FUNCTION_BLOCK PUBLIC PAEScaleGravimetric EXTENDS PAEScaleBase IMPLEMENTS IPAScaleGravimetric
VAR_INPUT
END_VAR
VAR_OUTPUT
END_VAR
VAR
	_CalmingTime : TIME;
	_CalmingWeight : LREAL;
	_IsDischarging : BOOL;
	_IsManualDosing : BOOL;
	_IsTared : BOOL;
	_ReqZeroReset : BOOL;
	_ReqZeroSet : BOOL;
	_StoredTareWeight : LREAL;
	_TareWeight : LREAL;
	_ZeroSet : BOOL;
	_ReqIsTared : BOOL;
	_TareCounterReq : DINT;
	_ActualWeightExternal : LREAL;
	_TareCounterRes : DINT;
END_VAR

{attribute 'monitoring' := 'call'}
//{attribute 'TcRpcEnable'}
PROPERTY PUBLIC ActualWeightExternal : LREAL
GET
ActualWeightExternal := _ActualWeightExternal;
END_GET
SET
_ActualWeightExternal := ActualWeightExternal;
Root.OnPropertyChangedLReal(THIS^, 84, _ActualWeightExternal);
END_SET
END_PROPERTY

{attribute 'monitoring' := 'call'}
//{attribute 'TcRpcEnable'}
PROPERTY PUBLIC CalmingTime : TIME
GET // PUBLIC
CalmingTime := _CalmingTime;
END_GET
SET // PUBLIC
_CalmingTime := CalmingTime;
Root.OnPropertyChangedTime(THIS^, 72, _CalmingTime);
END_SET
END_PROPERTY

{attribute 'monitoring' := 'call'}
//{attribute 'TcRpcEnable'}
PROPERTY CalmingWeight : LREAL
GET
CalmingWeight := _CalmingWeight;
END_GET
SET
_CalmingWeight := CalmingWeight;
Root.OnPropertyChangedLReal(THIS^, 73, _CalmingWeight);
END_SET
END_PROPERTY

METHOD FB_postinit
VAR_INPUT
	root : IACVariobatch;
END_VAR
SUPER^.FB_postinit(root);
root.OnPropertyChangedTime(THIS^, 72, _CalmingTime);
root.OnPropertyChangedLReal(THIS^, 73, _CalmingWeight);
root.OnPropertyChangedBool(THIS^,74, _ReqZeroSet);
root.OnPropertyChangedBool(THIS^, 75, _ReqZeroReset);
root.OnPropertyChangedLReal(THIS^, 76, _TareWeight);
root.OnPropertyChangedLReal(THIS^, 77, _StoredTareWeight);
root.OnPropertyChangedBool(THIS^, 78, _IsDischarging);
root.OnPropertyChangedBool(THIS^, 79, _IsTared);
root.OnPropertyChangedBool(THIS^, 80, _ZeroSet);
root.OnPropertyChangedBool(THIS^, 81, _IsManualDosing);
root.OnPropertyChangedBool(THIS^, 82, _ReqIsTared);
root.OnPropertyChangedDInt(THIS^, 83, _TareCounterReq);
root.OnPropertyChangedLReal(THIS^, 84, _ActualWeightExternal);
root.OnPropertyChangedDInt(THIS^, 85, _TareCounterRes);
END_METHOD

METHOD PUBLIC InvokeSetterBool
VAR_INPUT
	PropertyID : INT;
	PropertyValue : BOOL;
END_VAR
SUPER^.InvokeSetterBool(PropertyID, PropertyValue);
CASE PropertyID OF
	74:
		ReqZeroSet := PropertyValue;
	75:
		ReqZeroReset := PropertyValue;
	78:
		IsDischarging := PropertyValue;
	79:
		IsTared := PropertyValue;
	80:
		ZeroSet := PropertyValue;
	81:
		IsManualDosing := PropertyValue;
	82:
		ReqIsTared := PropertyValue;
END_CASE
END_METHOD

METHOD PUBLIC InvokeSetterDInt
VAR_INPUT
	PropertyID : INT;
	PropertyValue : DINT;
END_VAR
SUPER^.InvokeSetterDInt(PropertyID, PropertyValue);
CASE PropertyID OF
	83:
		TareCounterReq := PropertyValue;
	85:
		TareCounterRes := PropertyValue;
END_CASE
END_METHOD

METHOD PUBLIC InvokeSetterLReal
VAR_INPUT
	PropertyID : INT;
	PropertyValue : LREAL;
END_VAR
SUPER^.InvokeSetterLReal(PropertyID, PropertyValue);
CASE PropertyID OF
	73:
		CalmingWeight := PropertyValue;
	76:
		TareWeight := PropertyValue;
	77:
		StoredTareWeight := PropertyValue;
	84:
		ActualWeightExternal := PropertyValue;
END_CASE
END_METHOD

METHOD PUBLIC InvokeSetterTime
VAR_INPUT
	PropertyID : INT;
	PropertyValue : DINT;
END_VAR
SUPER^.InvokeSetterTime(PropertyID, PropertyValue);
CASE PropertyID OF 
	72:
		CalmingTime := TO_TIME(PropertyValue);
END_CASE
END_METHOD

{attribute 'monitoring' := 'call'}
//{attribute 'TcRpcEnable'}
PROPERTY PUBLIC IsDischarging : BOOL
GET // PUBLIC
IsDischarging := _IsDischarging;
END_GET
SET // PUBLIC
_IsDischarging := IsDischarging;
Root.OnPropertyChangedBool(THIS^, 78, _IsDischarging);
END_SET
END_PROPERTY

METHOD PUBLIC IsEnabledResetZero : BOOL
VAR_INPUT
END_VAR
END_METHOD

METHOD PUBLIC IsEnabledSetZero : BOOL
VAR_INPUT
END_VAR
END_METHOD

{attribute 'monitoring' := 'call'}
//{attribute 'TcRpcEnable'}
PROPERTY PUBLIC IsManualDosing : BOOL
GET // PUBLIC
IsManualDosing := _IsManualDosing;
END_GET
SET // PUBLIC
_IsManualDosing := IsManualDosing;
Root.OnPropertyChangedBool(THIS^, 81, _IsManualDosing);
END_SET
END_PROPERTY

{attribute 'monitoring' := 'call'}
//{attribute 'TcRpcEnable'}
PROPERTY PUBLIC IsTared : BOOL
GET // PUBLIC
IsTared := _IsTared;
END_GET
SET // PUBLIC
_IsTared := IsTared;
Root.OnPropertyChangedBool(THIS^, 79, _IsTared);
END_SET
END_PROPERTY

METHOD OnInitMemory
VAR_INPUT
	root : IACVariobatch;
END_VAR
RegisterProperty(root, 72, GCL.cSizeTIME); //CalmingTime
RegisterProperty(root, 73, GCL.cSizeLREAL); //CalmingWeight
RegisterProperty(root, 74, GCL.cSizeBYTE); //ReqZeroSet
RegisterProperty(root, 75, GCL.cSizeBYTE); //ReqZeroReset
RegisterProperty(root, 76, GCL.cSizeLREAL); //TareWeight
RegisterProperty(root, 77, GCL.cSizeLREAL); //StoredTaredWeight
RegisterProperty(root, 78, GCL.cSizeBYTE); //IsDischarging
RegisterProperty(root, 79, GCL.cSizeBYTE); //IsTared
RegisterProperty(root, 80, GCL.cSizeBYTE); //ZeroSet
RegisterProperty(root, 81, GCL.cSizeBYTE); //IsManualDosing
RegisterProperty(root, 82, GCL.cSizeBYTE); //ReqIsTared
RegisterProperty(root, 83, GCL.cSizeDINT); //TareCounterReq
RegisterProperty(root, 84, GCL.cSizeLREAL); //ActualWeightExternal
RegisterProperty(root, 85, GCL.cSizeDINT); //TareCounterRes
SUPER^.OnInitMemory(root);
END_METHOD

{attribute 'monitoring' := 'call'}
//{attribute 'TcRpcEnable'}
PROPERTY PUBLIC ReqIsTared : BOOL
GET
ReqIsTared := _ReqIsTared;
END_GET
SET // PUBLIC
_ReqIsTared := ReqIsTared;
Root.OnPropertyChangedBool(THIS^, 82, _ReqIsTared);
END_SET
END_PROPERTY

{attribute 'monitoring' := 'call'}
//{attribute 'TcRpcEnable'}
PROPERTY PUBLIC ReqZeroReset : BOOL
GET // PUBLIC
ReqZeroReset := _ReqZeroReset;
END_GET
SET // PUBLIC
_ReqZeroReset := ReqZeroReset;	
Root.OnPropertyChangedBool(THIS^, 75, _ReqZeroReset);
END_SET
END_PROPERTY

{attribute 'monitoring' := 'call'}
//{attribute 'TcRpcEnable'}
PROPERTY PUBLIC ReqZeroSet : BOOL
GET // PUBLIC
ReqZeroSet := _ReqZeroSet;
END_GET
SET // PUBLIC
_ReqZeroSet := ReqZeroSet;	
Root.OnPropertyChangedBool(THIS^,74, _ReqZeroSet);
END_SET
END_PROPERTY

METHOD PUBLIC ResetZero
VAR_INPUT
END_VAR
END_METHOD

METHOD PUBLIC SetZero
VAR_INPUT
END_VAR
END_METHOD

{attribute 'monitoring' := 'call'}
//{attribute 'TcRpcEnable'}
PROPERTY PUBLIC StoredTareWeight : LREAL
GET // PUBLIC
StoredTareWeight := _StoredTareWeight;
END_GET
SET // PUBLIC
_StoredTareWeight := StoredTareWeight;
Root.OnPropertyChangedLReal(THIS^, 77, _StoredTareWeight);
END_SET
END_PROPERTY

{attribute 'monitoring' := 'call'}
//{attribute 'TcRpcEnable'}
PROPERTY PUBLIC TareCounterReq : DINT
GET
TareCounterReq := _TareCounterReq;
END_GET
SET
_TareCounterReq := TareCounterReq;
Root.OnPropertyChangedDInt(THIS^, 83, _TareCounterReq);
END_SET
END_PROPERTY

{attribute 'monitoring' := 'call'}
//{attribute 'TcRpcEnable'}
PROPERTY PUBLIC TareCounterRes : DINT
GET
TareCounterRes := _TareCounterRes;
END_GET
SET
_TareCounterRes := TareCounterRes;
Root.OnPropertyChangedDInt(THIS^, 85, _TareCounterRes);
END_SET
END_PROPERTY

{attribute 'monitoring' := 'call'}
//{attribute 'TcRpcEnable'}
PROPERTY PUBLIC TareWeight : LREAL
GET // PUBLIC
TareWeight := _TareWeight;
END_GET
SET // PUBLIC
_TareWeight := TareWeight;
Root.OnPropertyChangedLReal(THIS^, 76, _TareWeight);
END_SET
END_PROPERTY

{attribute 'monitoring' := 'call'}
//{attribute 'TcRpcEnable'}
PROPERTY PUBLIC ZeroSet : BOOL
GET // PUBLIC
ZeroSet := _ZeroSet;
END_GET
SET // PUBLIC
_ZeroSet := ZeroSet;
Root.OnPropertyChangedBool(THIS^, 80, _ZeroSet);
END_SET
END_PROPERTY

END_FUNCTION_BLOCK

(* stored: Version 1.1.0.1, ProductVersion 3.1.4024.12
   POU PAEScaleGravimetric: Id {2689bd4b-c758-47c9-b36a-a0290e7a3511}, SpecialFunc None
   Property ActualWeightExternal: Id {e25f7741-07b2-46fd-9687-c860ee1a1068}
   Get Get: Id {18189f82-5514-4c61-a53c-0932185c160e}
   Set Set: Id {4b10a11c-d41f-41ce-b739-58d83de11f01}
   Property CalmingTime: Id {03837b69-0765-4d97-ac71-968db9750d03}
   Get Get: Id {3d1381dd-94dd-4102-91e2-361ccee45a82}
   Set Set: Id {fdef0714-f469-4235-98ee-4d98240d9990}
   Property CalmingWeight: Id {54282896-1f07-47cd-91c7-7650e7e99f26}
   Get Get: Id {1b726460-df51-4354-9026-1c6ae8026981}
   Set Set: Id {e2ca8723-2e5c-4e0c-9198-3ae122d26dfe}
   Method FB_postinit: Id {6ce4865d-e114-4d4e-a805-6cea694b7ddd}
   Method InvokeSetterBool: Id {bbf839f1-a3a9-4227-8116-4ea97104f046}
   Method InvokeSetterDInt: Id {a5ad1fd4-4132-4ccb-8b42-cf072c7bc429}
   Method InvokeSetterLReal: Id {cf72ab2a-6209-417a-bb23-6179e2b22e3f}
   Method InvokeSetterTime: Id {def87042-584f-44b1-b4d4-483d88e713d5}
   Property IsDischarging: Id {950ba824-8cbd-44a0-98ce-838c9f362ab1}
   Get Get: Id {12b04c7e-86c9-4ade-b3c0-1579d52867cb}
   Set Set: Id {474a4ebe-2e3a-461b-a0a0-d0a29dc98a25}
   Method IsEnabledResetZero: Id {c81e55c7-ece9-4fa4-b04f-181a6d7d85c6}
   Method IsEnabledSetZero: Id {dd8dcb68-0ca8-46ef-9a91-05afeaa9faee}
   Property IsManualDosing: Id {47777a7e-dfff-40d6-8a54-557154b22f2a}
   Get Get: Id {828f0136-b81a-4e57-b347-6dffa5657b4e}
   Set Set: Id {7b928f91-da61-48c0-8ca0-e9d7db920195}
   Property IsTared: Id {535d1c86-4f6a-4f74-8496-bc3721fb1984}
   Get Get: Id {9950b043-3209-4161-bfd4-6a61a5607243}
   Set Set: Id {19bcbf19-3414-415a-8f6d-c4c1feac517a}
   Method OnInitMemory: Id {cf13ca5c-7e40-4b4f-9cce-5c695fc15e03}
   Property ReqIsTared: Id {9fa7ddf8-aaad-431e-8ee7-1b4e25a9e236}
   Get Get: Id {032237ff-2cd9-4e20-b7a0-36255aa7e10d}
   Set Set: Id {421806d8-ead7-4fe9-9c76-1c2fd8f6339f}
   Property ReqZeroReset: Id {668329f0-9ef4-4912-b589-7bb8c4802a88}
   Get Get: Id {b98fbc6a-fac7-46ab-81c5-059d959cd7a2}
   Set Set: Id {ac3c66a3-f795-4ce4-8a29-17f75a46023d}
   Property ReqZeroSet: Id {c7d34542-4ec8-4c48-bd68-628b771f280a}
   Get Get: Id {738dd903-ff9d-4148-86a6-81ef0f7fab7c}
   Set Set: Id {e35f8501-0dab-4a10-abce-db723cb73ab4}
   Method ResetZero: Id {73c76d66-917f-4d7e-8b04-a989916a4d92}
   Method SetZero: Id {3b4cfb95-3d55-46b1-86ef-96f64e2143e2}
   Property StoredTareWeight: Id {ad0bcff8-4376-43b4-b735-78fd68263a81}
   Get Get: Id {d1f6c9b3-6837-4cad-bd0c-e2880666a5e7}
   Set Set: Id {f4764ea2-8fed-4178-a597-4acdaf951b33}
   Property TareCounterReq: Id {c81913b2-b7a2-444b-a589-ba9d873193e8}
   Get Get: Id {3c39aaf9-2a5e-4eaa-a618-1522cc4f5655}
   Set Set: Id {13ba6ed6-e8ed-4d15-9edf-ebbe9b1f7b47}
   Property TareCounterRes: Id {ae7b7d24-47ad-486d-bff8-fe81c0ff929a}
   Get Get: Id {a5859536-68c6-48c9-b628-6114a8e1244d}
   Set Set: Id {07df4e7b-82b3-4523-9993-bc40b5912021}
   Property TareWeight: Id {4518311c-984a-4703-9e1f-7190aec24180}
   Get Get: Id {cc9dc880-68fd-4d31-a303-b57ad2cb5b9a}
   Set Set: Id {f5cde28c-952a-40b1-82f2-f49949a872b4}
   Property ZeroSet: Id {4b012830-84ba-4039-9e7d-3ae3c477337e}
   Get Get: Id {69f2e0e3-fabc-4cef-b4da-f3985e788b61}
   Set Set: Id {f79884b8-e707-4111-9962-89a76ee73056} *)
